Universal Robots PolyScope program: 3exMove.urp

Program 3exMove (installation=default directory=/home/ur/ursim-current/programs createdIn=5.11.8.1010444 lastSavedIn=5.11.8.1010444 robotSerialNumber=20195399999)
Calibrated DH parameters: a=[0, -0.24355, -0.2132, 0, 0, 0]; d=[0.15185, 0, 0, 0.13105, 0.08535, 0.0921]; alpha=[1.570796, 0, 0, 1.570796, -1.570796, 0]; deltaTheta=[0, 0, 0, 0, 0, 0]
BeforeStart
  Script file /home/ur/ursim-current/programs/Script/4_Ex_Move.script
    | def Move(x, y, z, rx, ry, rz):
    | 	movel(p[x, y, z, rx, ry, rz], a=1, v=1)
    | 	sleep(1.0)
    | 	x = x + 0.01
    | 	y = y + 0.01
    | 	z = z + 0.01
    | 	movel(p[x, y, z, rx, ry, rz], a=1, v=1)
    | 	sleep(1.0)
    | end
Robot Program (runOnlyOnce=false)
  Wait Sleep waitTime=0.01
  x := 0.0
  y := 0.3
  z := 0.3
  rx := 0
  ry := 3.14
  rz := 0
  Script: Move(x,y,z,rx,ry,rz)
